// TIA Portal V17 program export: 0 tag tables, 0 data types, 3 data blocks, 14 code blocks (in call order from the OBs), 0 instance data blocks

DATA_BLOCK "DB_Params"   // DB70
{ S7_Optimized_Access := 'TRUE' }
VERSION : 0.1
// stored: AutoNumber false, DBAccessibleFromOPCUA true, IsOnlyStoredInLoadMemory false, IsRetainMemResEnabled false, IsWriteProtectedInAS false, MemoryReserve 100
   VAR
      SensorAngle : Real;   // angle absolu donné par capteur position [Rad]
      SensorAngleOffset : Real;   // Pour les capteurs 1 tour = pi / pour les capteurs 8 tours = 8*pi
      PinionModule : Real;   // Module pinion capteur pos [m] (std actuel : 3e-3)
      PinionTeethNum : Real;   // Nombre de dents du pinion (std actuel : 15)
   END_VAR
BEGIN
END_DATA_BLOCK

DATA_BLOCK "DB_Results"   // DB71
{ S7_Optimized_Access := 'TRUE' }
VERSION : 0.1
// stored: AutoNumber false, DBAccessibleFromOPCUA true, IsOnlyStoredInLoadMemory false, IsRetainMemResEnabled false, IsWriteProtectedInAS false, MemoryReserve 100
   VAR
      CylPosRes : Real;
      CylPosTpAngleRes : Real;
   END_VAR
BEGIN
END_DATA_BLOCK

DATA_BLOCK "projectParam"   // DB1
{ S7_Optimized_Access := 'TRUE' }
VERSION : 0.1
// stored: AutoNumber true, DBAccessibleFromOPCUA true, IsOnlyStoredInLoadMemory false, IsRetainMemResEnabled false, IsWriteProtectedInAS false, MemoryReserve 100
   VAR
      armParams : Array[1..3] of "typeArmParam";
   END_VAR
BEGIN
   armParams[1..3].armType := 'RCMA';
   armParams[1..3].armGeom.outLength := 8.839;
   armParams[1..3].armGeom.inLength := 9.449;
   armParams[1..3].armGeom.brHeight := 10.47;
   armParams[2].armGeom.brWidth := 10.47;
   armParams[1].motionControlParam.angleInputParam.filterTimeConsts[1..3] := 0.1;
   armParams[2].motionControlParam.angleInputParam.filterTimeConsts[1..3] := 0.1;
   armParams[3].motionControlParam.angleInputParam.filterTimeConsts[1..3] := 0.1;
   armParams[1].motionControlParam.angleInputParam.scalingParams[1].axisNum := 1;
   armParams[1].motionControlParam.angleInputParam.scalingParams[2].axisNum := 2;
   armParams[1].motionControlParam.angleInputParam.scalingParams[3].axisNum := 3;
   armParams[2].motionControlParam.angleInputParam.scalingParams[1].axisNum := 1;
   armParams[2].motionControlParam.angleInputParam.scalingParams[2].axisNum := 2;
   armParams[2].motionControlParam.angleInputParam.scalingParams[3].axisNum := 3;
   armParams[3].motionControlParam.angleInputParam.scalingParams[1].axisNum := 1;
   armParams[3].motionControlParam.angleInputParam.scalingParams[2].axisNum := 2;
   armParams[3].motionControlParam.angleInputParam.scalingParams[3].axisNum := 3;
   armParams[1].motionControlParam.angleInputParam.scalingParams[1..3]."a" := 1.0;
   armParams[2].motionControlParam.angleInputParam.scalingParams[1..3]."a" := 1.0;
   armParams[3].motionControlParam.angleInputParam.scalingParams[1..3]."a" := 1.0;
   armParams[1].motionControlParam.remoteInputParam.easyScalingParams[1].axisNum := 1;
   armParams[1].motionControlParam.remoteInputParam.easyScalingParams[2].axisNum := 2;
   armParams[1].motionControlParam.remoteInputParam.easyScalingParams[3].axisNum := 3;
   armParams[2].motionControlParam.remoteInputParam.easyScalingParams[1].axisNum := 1;
   armParams[2].motionControlParam.remoteInputParam.easyScalingParams[2].axisNum := 2;
   armParams[2].motionControlParam.remoteInputParam.easyScalingParams[3].axisNum := 3;
   armParams[3].motionControlParam.remoteInputParam.easyScalingParams[1].axisNum := 1;
   armParams[3].motionControlParam.remoteInputParam.easyScalingParams[2].axisNum := 2;
   armParams[3].motionControlParam.remoteInputParam.easyScalingParams[3].axisNum := 3;
   armParams[1].motionControlParam.remoteInputParam.easyScalingParams[1..3]."a" := 1.0;
   armParams[2].motionControlParam.remoteInputParam.easyScalingParams[1..3]."a" := 1.0;
   armParams[3].motionControlParam.remoteInputParam.easyScalingParams[1..3]."a" := 1.0;
   armParams[1].motionControlParam.remoteInputParam.convScalingParams[1].axisNum := 1;
   armParams[1].motionControlParam.remoteInputParam.convScalingParams[2].axisNum := 2;
   armParams[1].motionControlParam.remoteInputParam.convScalingParams[3].axisNum := 3;
   armParams[2].motionControlParam.remoteInputParam.convScalingParams[1].axisNum := 1;
   armParams[2].motionControlParam.remoteInputParam.convScalingParams[2].axisNum := 2;
   armParams[2].motionControlParam.remoteInputParam.convScalingParams[3].axisNum := 3;
   armParams[3].motionControlParam.remoteInputParam.convScalingParams[1].axisNum := 1;
   armParams[3].motionControlParam.remoteInputParam.convScalingParams[2].axisNum := 2;
   armParams[3].motionControlParam.remoteInputParam.convScalingParams[3].axisNum := 3;
   armParams[1].motionControlParam.remoteInputParam.convScalingParams[1..3]."a" := 1.0;
   armParams[2].motionControlParam.remoteInputParam.convScalingParams[1..3]."a" := 1.0;
   armParams[3].motionControlParam.remoteInputParam.convScalingParams[1..3]."a" := 1.0;
   armParams[1].motionControlParam.remoteInputParam.filterTimeConsts[1..3] := 0.1;
   armParams[2].motionControlParam.remoteInputParam.filterTimeConsts[1..3] := 0.1;
   armParams[3].motionControlParam.remoteInputParam.filterTimeConsts[1..3] := 0.1;
   armParams[1].motionControlParam.angularSpeedGains[1..3] := 0.018;
   armParams[2].motionControlParam.angularSpeedGains[1..3] := 0.018;
   armParams[3].motionControlParam.angularSpeedGains[1..3] := 0.018;
   armParams[1].motionControlParam.cartSpeedGains[1..3] := 0.15;
   armParams[2].motionControlParam.cartSpeedGains[1..3] := 0.15;
   armParams[3].motionControlParam.cartSpeedGains[1..3] := 0.15;
   armParams[1].motionControlParam.regulParams[1..3].fOn := 1.0;
   armParams[2].motionControlParam.regulParams[1..3].fOn := 1.0;
   armParams[3].motionControlParam.regulParams[1..3].fOn := 1.0;
   armParams[1].motionControlParam.regulParams[1..3].pOn := 1.0;
   armParams[2].motionControlParam.regulParams[1..3].pOn := 1.0;
   armParams[3].motionControlParam.regulParams[1..3].pOn := 1.0;
   armParams[1].motionControlParam.regulParams[1..3].kP := 0.001;
   armParams[2].motionControlParam.regulParams[1..3].kP := 0.001;
   armParams[3].motionControlParam.regulParams[1..3].kP := 0.001;
   armParams[1].motionControlParam.regulParams[1..3].tI := 0.1;
   armParams[2].motionControlParam.regulParams[1..3].tI := 0.1;
   armParams[3].motionControlParam.regulParams[1..3].tI := 0.1;
   armParams[1].motionControlParam.regulParams[1..3].tD := 0.1;
   armParams[2].motionControlParam.regulParams[1..3].tD := 0.1;
   armParams[3].motionControlParam.regulParams[1..3].tD := 0.1;
   armParams[1].motionControlParam.outputParam.filterTimeConsts[1..3] := 0.1;
   armParams[2].motionControlParam.outputParam.filterTimeConsts[1..3] := 0.1;
   armParams[3].motionControlParam.outputParam.filterTimeConsts[1..3] := 0.1;
   armParams[1..3].motionControlParam.satParam.deltaSatGainNeg := 0.01;
   armParams[1].motionControlParam.satParam.satLevels[1..2] := 1.0;
   armParams[1].motionControlParam.satParam.satLevels[3] := 0.5;
   armParams[2].motionControlParam.satParam.satLevels[1..2] := 1.0;
   armParams[2].motionControlParam.satParam.satLevels[3] := 0.5;
   armParams[3].motionControlParam.satParam.satLevels[1..2] := 1.0;
   armParams[3].motionControlParam.satParam.satLevels[3] := 0.5;
   armParams[1..3].motionControlParam.minSetpoint := 0.05;
   armParams[1..3].motionControlParam.minSpeed := 0.01;
   armParams[1].axisParams[1].axisType := 'direct';
   armParams[1].axisParams[2].axisType := 'double';
   armParams[1].axisParams[3].axisType := 'sheave';
   armParams[2].axisParams[1].axisType := 'direct';
   armParams[2].axisParams[2].axisType := 'double';
   armParams[2].axisParams[3].axisType := 'sheave';
   armParams[3].axisParams[1].axisType := 'direct';
   armParams[3].axisParams[2].axisType := 'double';
   armParams[3].axisParams[3].axisType := 'sheave';
   armParams[1].axisParams[1].cylinderType := 'diff';
   armParams[1].axisParams[2..3].cylinderType := 'sym';
   armParams[2].axisParams[1].cylinderType := 'diff';
   armParams[2].axisParams[2..3].cylinderType := 'sym';
   armParams[3].axisParams[1].cylinderType := 'diff';
   armParams[3].axisParams[2..3].cylinderType := 'sym';
   armParams[1].axisParams[1..3].cylinderDir := 1.0;
   armParams[2].axisParams[1..3].cylinderDir := 1.0;
   armParams[3].axisParams[1..3].cylinderDir := 1.0;
   armParams[1].axisParams[1].pistonDiam := 0.1;
   armParams[1].axisParams[2].pistonDiam := 0.14;
   armParams[1].axisParams[3].pistonDiam := 0.11;
   armParams[2].axisParams[1].pistonDiam := 0.1;
   armParams[2].axisParams[2].pistonDiam := 0.14;
   armParams[2].axisParams[3].pistonDiam := 0.11;
   armParams[3].axisParams[1].pistonDiam := 0.1;
   armParams[3].axisParams[2].pistonDiam := 0.14;
   armParams[3].axisParams[3].pistonDiam := 0.11;
   armParams[1].axisParams[1].rodDiam := 0.045;
   armParams[1].axisParams[2].rodDiam := 0.065;
   armParams[1].axisParams[3].rodDiam := 0.055;
   armParams[2].axisParams[1].rodDiam := 0.045;
   armParams[2].axisParams[2].rodDiam := 0.065;
   armParams[2].axisParams[3].rodDiam := 0.055;
   armParams[3].axisParams[1].rodDiam := 0.045;
   armParams[3].axisParams[2].rodDiam := 0.065;
   armParams[3].axisParams[3].rodDiam := 0.055;
   armParams[1].axisParams[1].stroke := 0.62;
   armParams[1].axisParams[2].stroke := 1.4;
   armParams[1].axisParams[3].stroke := 1.0;
   armParams[2].axisParams[1].stroke := 0.62;
   armParams[2].axisParams[2].stroke := 1.4;
   armParams[2].axisParams[3].stroke := 1.0;
   armParams[3].axisParams[1].stroke := 0.62;
   armParams[3].axisParams[2].stroke := 1.4;
   armParams[3].axisParams[3].stroke := 1.0;
   armParams[1].axisParams[1].rodPivotPos[1] := 0.435;
   armParams[1].axisParams[1].rodPivotPos[2] := 0.05;
   armParams[2].axisParams[1].rodPivotPos[1] := 0.435;
   armParams[2].axisParams[1].rodPivotPos[2] := 0.05;
   armParams[3].axisParams[1].rodPivotPos[1] := 0.435;
   armParams[3].axisParams[1].rodPivotPos[2] := 0.05;
   armParams[1].axisParams[1].bodyPivotPos[1] := 0.224;
   armParams[1].axisParams[1].bodyPivotPos[2] := 0.775;
   armParams[2].axisParams[1].bodyPivotPos[1] := 0.224;
   armParams[2].axisParams[1].bodyPivotPos[2] := 0.775;
   armParams[3].axisParams[1].bodyPivotPos[1] := 0.224;
   armParams[3].axisParams[1].bodyPivotPos[2] := 0.775;
   armParams[1].axisParams[1].movingCylinder := TRUE;
   armParams[2].axisParams[1].movingCylinder := TRUE;
   armParams[3].axisParams[1].movingCylinder := TRUE;
   armParams[1].axisParams[1..3].presDrop := 1000000.0;
   armParams[2].axisParams[1..3].presDrop := 1000000.0;
   armParams[3].axisParams[1..3].presDrop := 1000000.0;
   armParams[1].axisParams[1].nomFlow := 1.67E-05;
   armParams[1].axisParams[2].nomFlow := 0.00013;
   armParams[1].axisParams[3].nomFlow := 7.5E-05;
   armParams[2].axisParams[1].nomFlow := 1.67E-05;
   armParams[2].axisParams[2].nomFlow := 0.00013;
   armParams[2].axisParams[3].nomFlow := 7.5E-05;
   armParams[3].axisParams[1].nomFlow := 1.67E-05;
   armParams[3].axisParams[2].nomFlow := 0.00013;
   armParams[3].axisParams[3].nomFlow := 7.5E-05;
   armParams[1].axisParams[1..3].setpointJump := 0.2;
   armParams[2].axisParams[1..3].setpointJump := 0.2;
   armParams[3].axisParams[1..3].setpointJump := 0.2;
   armParams[1].axisParams[1..3].setpointMin := 0.01;
   armParams[2].axisParams[1..3].setpointMin := 0.01;
   armParams[3].axisParams[1..3].setpointMin := 0.01;
   armParams[1].axisParams[2].sheaveDiam := 1.0;
   armParams[1].axisParams[3].sheaveDiam := 0.82;
   armParams[2].axisParams[2].sheaveDiam := 1.0;
   armParams[2].axisParams[3].sheaveDiam := 0.82;
   armParams[3].axisParams[2].sheaveDiam := 1.0;
   armParams[3].axisParams[3].sheaveDiam := 0.82;
   armParams[1].axisParams[1..3].naturalFrequency := 2.0;
   armParams[2].axisParams[1..3].naturalFrequency := 2.0;
   armParams[3].axisParams[1..3].naturalFrequency := 2.0;
   armParams[1].axisParams[1..3].damping := 0.2;
   armParams[2].axisParams[1..3].damping := 0.2;
   armParams[3].axisParams[1..3].damping := 0.2;
END_DATA_BLOCK

ORGANIZATION_BLOCK "Main"   // OB1, LAD, ProgramCycle
TITLE = "Main Program Sweep (Cycle)"
{ S7_Optimized_Access := 'TRUE' }
VERSION : 0.1
// stored: AutoNumber true, IsIECCheckEnabled false, SetENOAutomatically false
   VAR_INPUT
      Initial_Call : Bool;   // Initial call of this OB
      Remanence : Bool;   // =True, if remanent data are available
   END_VAR
BEGIN

REGION Network 1: Call functions & Subfonctions
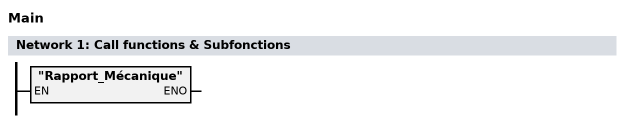
   RUNG wire#powerrail
      "Rapport_Mécanique"()
   END_RUNG
   // the same network as SCL:
   "Rapport_Mécanique"();
END_REGION
END_ORGANIZATION_BLOCK

FUNCTION "Rapport_Mécanique" : Void   // FC70, LAD
{ S7_Optimized_Access := 'TRUE' }
VERSION : 0.1
// stored: AutoNumber false, IsIECCheckEnabled false, SetENOAutomatically false, UDAEnableTagReadback false
BEGIN

REGION Network 1: Test du bloc CylPos
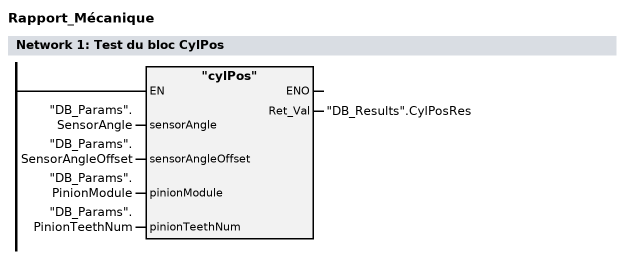
   RUNG wire#powerrail
      "cylPos"(sensorAngle := "DB_Params".SensorAngle, sensorAngleOffset := "DB_Params".SensorAngleOffset, pinionModule := "DB_Params".PinionModule, pinionTeethNum := "DB_Params".PinionTeethNum, Ret_Val => "DB_Results".CylPosRes)
   END_RUNG
   // the same network as SCL:
   "DB_Results".CylPosRes := "cylPos"(sensorAngle := "DB_Params".SensorAngle,
                           sensorAngleOffset := "DB_Params".SensorAngleOffset,
                           pinionModule := "DB_Params".PinionModule,
                           pinionTeethNum := "DB_Params".PinionTeethNum);
END_REGION
END_FUNCTION

FUNCTION "cylPos" : Real
{ S7_Optimized_Access := 'TRUE' }
VERSION : 0.1
   VAR_INPUT 
      sensorAngle : Real;
      sensorAngleOffset : Real;
      pinionModule : Real;
      pinionTeethNum : Real;
   END_VAR


BEGIN
	(*Calcul de la variation relative de position du vérin à partir de la position médiane*)
	#cylPos := (#sensorAngle - #sensorAngleOffset) * #pinionModule * #pinionTeethNum;
END_FUNCTION

ORGANIZATION_BLOCK "Cyclic interrupt"   // OB30, LAD, CyclicInterrupt
{ S7_Optimized_Access := 'TRUE' }
VERSION : 0.1
// stored: AutoNumber true, IsIECCheckEnabled false, SetENOAutomatically false
   VAR_INPUT
      Initial_Call : Bool;   // Initial call of this OB
      Event_Count : Int;   // Events discarded
   END_VAR
BEGIN

REGION Network 1
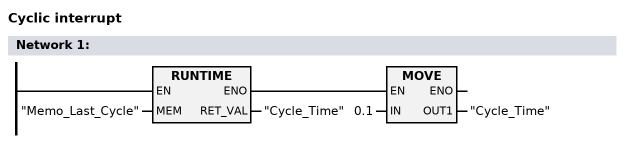
   // no SCL statement known for Runtime: written as a call
   // ENO of a box is taken as its EN; it also drops when the box reports an error
   "Cycle_Time" := Runtime(mem := "Memo_Last_Cycle");
   "Cycle_Time" := 0.1;
END_REGION
END_ORGANIZATION_BLOCK

ORGANIZATION_BLOCK "Diagnostic error interrupt"   // OB82, LAD, DiagnosticErrorInterrupt
{ S7_Optimized_Access := 'TRUE' }
VERSION : 0.1
// stored: IsIECCheckEnabled false, SetENOAutomatically false
   VAR_INPUT
      IO_State : Word;   // IO state of the HW object
      LADDR : HW_ANY;   // Hardware identifier
      Channel : UInt;   // Channel number
      MultiError : Bool;   // =true if more than one error is present
   END_VAR
BEGIN
END_ORGANIZATION_BLOCK

ORGANIZATION_BLOCK "Main_with_Cycle"   // OB123, LAD, ProgramCycle
TITLE = "Main Program Sweep (Cycle)"
{ S7_Optimized_Access := 'TRUE' }
VERSION : 0.1
// stored: AutoNumber true, IsIECCheckEnabled false, SetENOAutomatically false
   VAR_INPUT
      Initial_Call : Bool;   // Initial call of this OB
      Remanence : Bool;   // =True, if remanent data are available
   END_VAR
BEGIN
END_ORGANIZATION_BLOCK

ORGANIZATION_BLOCK "Rack or station failure"   // OB86, LAD, RackOrStationFailure
{ S7_Optimized_Access := 'TRUE' }
VERSION : 0.1
// stored: IsIECCheckEnabled false, SetENOAutomatically false
   VAR_INPUT
      LADDR : HW_DEVICE;   // Hardware identifier
      Event_Class : Byte;   // Event class
      Fault_ID : Byte;   // Fault identifier
   END_VAR
BEGIN
END_ORGANIZATION_BLOCK

ORGANIZATION_BLOCK "Startup"   // OB100, LAD, Startup
TITLE = "Complete Restart"
{ S7_Optimized_Access := 'TRUE' }
VERSION : 0.1
// stored: AutoNumber true, IsIECCheckEnabled false, SetENOAutomatically false
   VAR_INPUT
      LostRetentive : Bool;   // True if retentive data are lost
      LostRTC : Bool;   // True if date and time are lost
   END_VAR
BEGIN

REGION Network 1: Appel FCxxxx
END_REGION
END_ORGANIZATION_BLOCK

FUNCTION "cylPosToAngle" : Real
{ S7_Optimized_Access := 'TRUE' }
VERSION : 0.1
   VAR_INPUT 
      cylPosRel : Real;
      Xp : Real;
      Yp : Real;
      Xv : Real;
      Yv : Real;
   END_VAR

   VAR_TEMP 
      Rv : Real;
      D0 : Real;
      phiV0 : Real;
      X1 : Real;
      X2 : Real;
      X3 : Real;
      SIN_PHI : Real;
      COS_PHI : Real;
   END_VAR


BEGIN
	(* Calcul de la position angulaire de la manoeuvre à partir de la position du vérin *)
	#Rv := SQRT((#Xv ** 2 + #Yv ** 2));
	#D0 := SQRT(((#Xp - #Xv) ** 2 + (#Yp - #Yv) ** 2));
	#phiV0 := ATAN(#Yv / #Xv);
	#X1 := 2 * #Rv * #Xp;
	#X2 := 2 * #Rv * #Yp;
	#X3 := #Xp ** 2 + #Yp ** 2 + #Rv ** 2 - (#D0 + #cylPosRel) ** 2;
	
	#SIN_PHI := (#X2 * #X3 + #X1 * SQRT((#X1 ** 2 + #X2 ** 2 - #X3 ** 2))) / (#X1 ** 2 + #X2 ** 2);
	#COS_PHI := (#X1 * #X3 - #X2 * SQRT((#X1 ** 2 + #X2 ** 2 - #X3 ** 2))) / (#X1 ** 2 + #X2 ** 2);
	
	#cylPosToAngle := "Atan2"("x" := #COS_PHI, "y" := #SIN_PHI) - #phiV0;
END_FUNCTION

FUNCTION "ConvTrajectoryPlan" : Void
{ S7_Optimized_Access := 'TRUE' }
FAMILY : EasyDrive
VERSION : 0.1
//Ancien block CON
   VAR_INPUT 
      setSpeeds : Array[1.."AXIS_NUM"] of Real;
      motionControlParam : "typeMotionControlParam";
   END_VAR

   VAR_OUTPUT 
      angleSpeeds : Array[1.."AXIS_NUM"] of Real;
   END_VAR

   VAR_TEMP 
      axisCounter : Int;
   END_VAR


BEGIN
	(* Trajectory calculation in conventionnal mode *)
	
	FOR #axisCounter := 1 TO "AXIS_NUM" DO
	    #angleSpeeds[#axisCounter] := #setSpeeds[#axisCounter] * #motionControlParam.angularSpeedGains[#axisCounter];
	END_FOR;
	
END_FUNCTION

FUNCTION "ForwardKinematicSimple" : Void
{ S7_Optimized_Access := 'TRUE' }
VERSION : 0.1
   VAR_INPUT 
      armGeom : "typeArmGeom";
      angles : Array[1..3] of Real;
   END_VAR

   VAR_OUTPUT 
      pos : Array[1..3] of Real;
   END_VAR

   VAR_TEMP 
      F : Real;
      G : Real;
      phi : Real;
      beta : Real;
      alpha : Real;
      H : Real;
   END_VAR


BEGIN
	(* Simple direct kinematic of the rotation n°4 *)
	
	(* Parameters retrieval *)
	#F := #armGeom.outLength;
	#G := #armGeom.inLength;
	#H := #armGeom.brHeight;
	#phi := #angles[1];
	#alpha := #angles[2];
	#beta := #angles[3];
	
	(* Axis x *)
	#pos[1] := SIN(#phi) * (#F * SIN(#beta) + #G * COS(#alpha));
	(* Axis y *)
	#pos[2] := - COS(#phi) * (#F * SIN(#beta) + #G * COS(#alpha));
	(* Axis z *)
	#pos[3] := - #F * COS(#beta) + #G * SIN(#alpha) + #H;
	
END_FUNCTION

FUNCTION "Sat" : Real
{ S7_Optimized_Access := 'TRUE' }
VERSION : 0.1
   VAR_INPUT 
      input : Real;
   END_VAR


BEGIN
	(* Calculate saturation of an input between -1.0 and 1.0 *)
	
	IF #input > 1.0 THEN
	    #Sat := 1.0;
	ELSIF #input < - 1.0 THEN
	    #Sat := -1.0;
	ELSE
	    #Sat := #input;
	END_IF;
	
END_FUNCTION

FUNCTION "Scaling" : Real
{ S7_Optimized_Access := 'TRUE' }
VERSION : 0.1
   VAR_INPUT 
      input : Real;
      scaleParam : "typeScaleParam";
   END_VAR


BEGIN
	
	(* Module for linear scaling : y = ax + b *)
	
	#Scaling := #scaleParam.a * #input + #scaleParam.b;
	
END_FUNCTION

FUNCTION_BLOCK "SetpointOutputs"
{ S7_Optimized_Access := 'TRUE' }
VERSION : 0.1
   VAR_INPUT 
      setpointProps : Array[1.."AXIS_NUM"] of Real;
      motionControlParam : "typeMotionControlParam";
      timeCycle : Real;
      axisParams : Array[1.."AXIS_NUM"] of "typeAxisParam";
   END_VAR

   VAR_OUTPUT 
      finalSetpointProps : Array[1.."AXIS_NUM"] of Real;
      sat : Bool;
   END_VAR

   VAR 
      InstFirstOrderFilters { S7_SetPoint := 'False'} : Array[1.."AXIS_NUM"] of "FirstOrderFilter";
   END_VAR

   VAR_TEMP 
      axisCounter : Int;
      aux : Array[1.."AXIS_NUM"] of Real;
      checkSatOutputs : Array[1.."AXIS_NUM"] of Bool;
      satOutputs : Array[1.."AXIS_NUM"] of Real;
      jumpOutputs : Array[1.."AXIS_NUM"] of Real;
   END_VAR


BEGIN
	(* Output process *)
	
	FOR #axisCounter := 1 TO "AXIS_NUM" DO
	    
	    #InstFirstOrderFilters[#axisCounter](input := #setpointProps[#axisCounter],
	                                         timeConstant := #motionControlParam.outputParam.filterTimeConsts[#axisCounter],
	                                         timeCycle := #timeCycle,
	                                         enable := TRUE,
	                                         output => #aux[#axisCounter]);
	    
	    #satOutputs[#axisCounter] := "Sat"(input := #aux[#axisCounter]);
	    
	    #finalSetpointProps[#axisCounter] := "Jump"(axisParam := #axisParams[#axisCounter],
	                                                input := #satOutputs[#axisCounter]);
	END_FOR;
	
	#sat := "CheckSat"(satParam := #motionControlParam.satParam, setpointProp := #aux);
	
	
END_FUNCTION_BLOCK
